// TIA Portal V20 export
ORGANIZATION_BLOCK "CyclicInterrupt"   // OB32, LAD, CyclicInterrupt
// stored: Namespace Unit1.Em3, SetENOAutomatically false
   VAR_INPUT
      Initial_Call : Bool;   // Initial call of this OB
      Event_Count : Int;   // Events discarded
   END_VAR
BEGIN

REGION Network 1
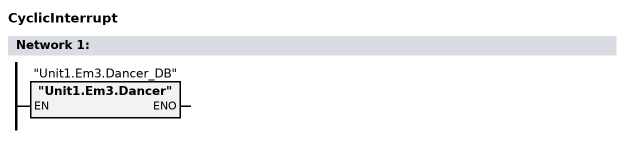
   RUNG wire#powerrail
      "Unit1.Em3.Dancer_DB"()
   END_RUNG
   // the same network as SCL:
   "Unit1.Em3.Dancer_DB"();   // "Unit1.Em3.Dancer"
END_REGION
END_ORGANIZATION_BLOCK
